ABB RAPID module: Module1_J.mod

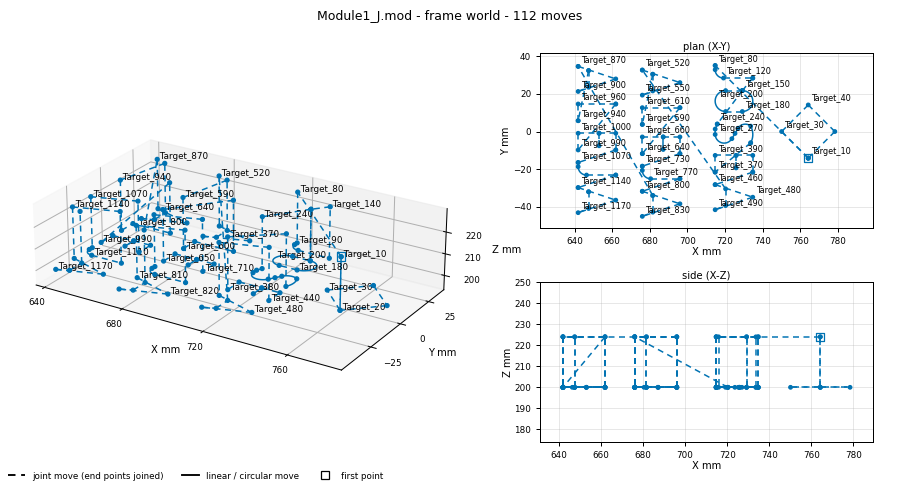
[picture p0: tool path of Module1_J.mod in frame world, 112 of 112 moves have a stored position in this frame; points joined in program order, loops and branches not executed]
MODULE Module1
!Definición de los puntos por donde pasa la trayectoria en forma de robtargets.
!
    CONST robtarget Target_10:=[[149.241,70.858,24],[0.130526196,0,0.991444861,0],[-1,1,-2,0],[9E+09,9E+09,9E+09,9E+09,9E+09,9E+09]];
    CONST robtarget Target_20:=[[149.241,70.858,0],[0.130526196,0,0.991444861,0],[-1,1,-2,0],[9E+09,9E+09,9E+09,9E+09,9E+09,9E+09]];
    CONST robtarget Target_30:=[[135.099,85,0],[0.130526196,0,0.991444861,0],[-1,1,-2,0],[9E+09,9E+09,9E+09,9E+09,9E+09,9E+09]];
    CONST robtarget Target_40:=[[149.241,99.142,0],[0.130526196,0,0.991444861,0],[0,2,-2,0],[9E+09,9E+09,9E+09,9E+09,9E+09,9E+09]];
    CONST robtarget Target_50:=[[163.384,85,0],[0.130526196,0,0.991444861,0],[0,2,-3,0],[9E+09,9E+09,9E+09,9E+09,9E+09,9E+09]];
    CONST robtarget Target_60:=[[149.241,70.858,0],[0.130526196,0,0.991444861,0],[0,2,-3,0],[9E+09,9E+09,9E+09,9E+09,9E+09,9E+09]];
    CONST robtarget Target_70:=[[149.241,70.858,24],[0.130526196,0,0.991444861,0],[-1,1,-2,0],[9E+09,9E+09,9E+09,9E+09,9E+09,9E+09]];
    CONST robtarget Target_80:=[[99.757,120.09,24],[0.130526201,0,0.99144486,-0.000000003],[-1,1,-2,0],[9E+09,9E+09,9E+09,9E+09,9E+09,9E+09]];
    CONST robtarget Target_90:=[[99.757,120.09,0],[0.130526201,0,0.99144486,-0.000000003],[0,2,-3,0],[9E+09,9E+09,9E+09,9E+09,9E+09,9E+09]];
    CONST robtarget Target_100:=[[99.757,117.868,0],[0.130526201,0,0.99144486,-0.000000003],[0,2,-3,0],[9E+09,9E+09,9E+09,9E+09,9E+09,9E+09]];
    CONST robtarget Target_110:=[[101.05812907,114.725008652,0.000349024],[0.130526181,-0.000000019,0.991444863,0.000000016],[0,2,-3,0],[9E+09,9E+09,9E+09,9E+09,9E+09,9E+09]];
    CONST robtarget Target_120:=[[104.201,113.423,0],[0.130526201,0,0.99144486,-0.000000003],[0,2,-3,0],[9E+09,9E+09,9E+09,9E+09,9E+09,9E+09]];
    CONST robtarget Target_130:=[[119.757,113.423,0],[0.130526201,0,0.99144486,-0.000000003],[0,2,-3,0],[9E+09,9E+09,9E+09,9E+09,9E+09,9E+09]];
    CONST robtarget Target_140:=[[119.757,113.423,24],[0.130526201,0,0.99144486,-0.000000003],[0,2,-3,0],[9E+09,9E+09,9E+09,9E+09,9E+09,9E+09]];
    CONST robtarget Target_150:=[[114.201,106.757,24],[0.130526201,0,0.99144486,-0.000000003],[0,2,-3,0],[9E+09,9E+09,9E+09,9E+09,9E+09,9E+09]];
    CONST robtarget Target_160:=[[114.201,106.757,0],[0.130526201,0,0.99144486,-0.000000003],[0,2,-3,0],[9E+09,9E+09,9E+09,9E+09,9E+09,9E+09]];
    CONST robtarget Target_170:=[[119.757,101.201,0],[0.130526201,0,0.99144486,-0.000000003],[0,2,-3,0],[9E+09,9E+09,9E+09,9E+09,9E+09,9E+09]];
    CONST robtarget Target_180:=[[114.201,95.645,0],[0.130526201,0,0.99144486,-0.000000003],[0,2,-3,0],[9E+09,9E+09,9E+09,9E+09,9E+09,9E+09]];
    CONST robtarget Target_190:=[[105.312,95.645,0],[0.130526201,0,0.99144486,-0.000000003],[0,2,-3,0],[9E+09,9E+09,9E+09,9E+09,9E+09,9E+09]];
    CONST robtarget Target_200:=[[99.757,101.201,0],[0.130526201,0,0.99144486,-0.000000003],[0,2,-3,0],[9E+09,9E+09,9E+09,9E+09,9E+09,9E+09]];
    CONST robtarget Target_210:=[[105.312,106.757,0],[0.130526201,0,0.99144486,-0.000000003],[0,2,-3,0],[9E+09,9E+09,9E+09,9E+09,9E+09,9E+09]];
    CONST robtarget Target_220:=[[114.201,106.757,0],[0.130526201,0,0.99144486,-0.000000003],[0,2,-3,0],[9E+09,9E+09,9E+09,9E+09,9E+09,9E+09]];
    CONST robtarget Target_230:=[[114.201,106.757,24],[0.130526201,0,0.99144486,-0.000000003],[0,2,-3,0],[9E+09,9E+09,9E+09,9E+09,9E+09,9E+09]];
    CONST robtarget Target_240:=[[100.868,88.979,24],[0.130526201,0,0.99144486,-0.000000003],[0,2,-3,0],[9E+09,9E+09,9E+09,9E+09,9E+09,9E+09]];
    CONST robtarget Target_250:=[[100.868,88.979,0],[0.130526201,0,0.99144486,-0.000000003],[0,2,-3,0],[9E+09,9E+09,9E+09,9E+09,9E+09,9E+09]];
    CONST robtarget Target_260:=[[99.766,86.31,0],[0.130526201,0,0.99144486,-0.000000003],[0,2,-3,0],[9E+09,9E+09,9E+09,9E+09,9E+09,9E+09]];
    CONST robtarget Target_270:=[[99.757,83.423,0],[0.130526201,0,0.99144486,-0.000000003],[0,2,-3,0],[9E+09,9E+09,9E+09,9E+09,9E+09,9E+09]];
    CONST robtarget Target_280:=[[103.37,78.987,0],[0.130526201,0,0.99144486,-0.000000003],[-1,1,-2,0],[9E+09,9E+09,9E+09,9E+09,9E+09,9E+09]];
    CONST robtarget Target_290:=[[108.646,81.201,0],[0.130526201,0,0.99144486,-0.000000003],[-1,1,-2,0],[9E+09,9E+09,9E+09,9E+09,9E+09,9E+09]];
    CONST robtarget Target_300:=[[110.312,83.979,0],[0.130526201,0,0.99144486,-0.000000003],[-1,1,-2,0],[9E+09,9E+09,9E+09,9E+09,9E+09,9E+09]];
    CONST robtarget Target_310:=[[111.979,86.757,0],[0.130526201,0,0.99144486,-0.000000003],[-1,1,-2,0],[9E+09,9E+09,9E+09,9E+09,9E+09,9E+09]];
    CONST robtarget Target_320:=[[115.054,88.861,0],[0.130526201,0,0.99144486,-0.000000003],[0,2,-3,0],[9E+09,9E+09,9E+09,9E+09,9E+09,9E+09]];
    CONST robtarget Target_340:=[[119.766,83.423,0],[0.130526201,0,0.99144486,-0.000000003],[0,2,-3,0],[9E+09,9E+09,9E+09,9E+09,9E+09,9E+09]];
    CONST robtarget Target_350:=[[118.646,78.979,0],[0.130526201,0,0.99144486,-0.000000003],[-1,1,-2,0],[9E+09,9E+09,9E+09,9E+09,9E+09,9E+09]];
    CONST robtarget Target_360:=[[118.646,78.979,24],[0.130526201,0,0.99144486,-0.000000003],[-1,1,-2,0],[9E+09,9E+09,9E+09,9E+09,9E+09,9E+09]];
    CONST robtarget Target_370:=[[99.757,63.423,24],[0.130526201,0,0.99144486,-0.000000003],[-1,1,-2,0],[9E+09,9E+09,9E+09,9E+09,9E+09,9E+09]];
    CONST robtarget Target_380:=[[99.757,63.423,0],[0.130526201,0,0.99144486,-0.000000003],[-1,1,-2,0],[9E+09,9E+09,9E+09,9E+09,9E+09,9E+09]];
    CONST robtarget Target_390:=[[99.757,72.312,0],[0.130526201,0,0.99144486,-0.000000003],[-1,1,-2,0],[9E+09,9E+09,9E+09,9E+09,9E+09,9E+09]];
    CONST robtarget Target_400:=[[110.868,72.312,0],[0.130526201,0,0.99144486,-0.000000003],[-1,1,-2,0],[9E+09,9E+09,9E+09,9E+09,9E+09,9E+09]];
    CONST robtarget Target_410:=[[110.868,65.645,0],[0.130526201,0,0.99144486,-0.000000003],[-1,1,-2,0],[9E+09,9E+09,9E+09,9E+09,9E+09,9E+09]];
    CONST robtarget Target_420:=[[110.868,72.312,0],[0.130526201,0,0.99144486,-0.000000003],[-1,1,-2,0],[9E+09,9E+09,9E+09,9E+09,9E+09,9E+09]];
    CONST robtarget Target_430:=[[119.757,72.312,0],[0.130526201,0,0.99144486,-0.000000003],[-1,1,-2,0],[9E+09,9E+09,9E+09,9E+09,9E+09,9E+09]];
    CONST robtarget Target_440:=[[119.757,63.423,0],[0.130526201,0,0.99144486,-0.000000003],[-1,1,-2,0],[9E+09,9E+09,9E+09,9E+09,9E+09,9E+09]];
    CONST robtarget Target_450:=[[119.757,63.423,24],[0.130526201,0,0.99144486,-0.000000003],[-1,1,-2,0],[9E+09,9E+09,9E+09,9E+09,9E+09,9E+09]];
    CONST robtarget Target_460:=[[99.757,56.757,24],[0.130526201,0,0.99144486,-0.000000003],[-1,1,-2,0],[9E+09,9E+09,9E+09,9E+09,9E+09,9E+09]];
    CONST robtarget Target_470:=[[99.757,56.757,0],[0.130526201,0,0.99144486,-0.000000003],[-1,1,-2,0],[9E+09,9E+09,9E+09,9E+09,9E+09,9E+09]];
    CONST robtarget Target_480:=[[119.757,50.09,0],[0.130526201,0,0.99144486,-0.000000003],[-1,1,-2,0],[9E+09,9E+09,9E+09,9E+09,9E+09,9E+09]];
    CONST robtarget Target_490:=[[99.757,43.423,0],[0.130526201,0,0.99144486,-0.000000003],[-1,1,-2,0],[9E+09,9E+09,9E+09,9E+09,9E+09,9E+09]];
    CONST robtarget Target_500:=[[105.312,45.645,0],[0.130526201,0,0.99144486,-0.000000003],[-1,1,-2,0],[9E+09,9E+09,9E+09,9E+09,9E+09,9E+09]];
    CONST robtarget Target_510:=[[105.312,54.534,0],[0.130526201,0,0.99144486,-0.000000003],[-1,1,-2,0],[9E+09,9E+09,9E+09,9E+09,9E+09,9E+09]];
    CONST robtarget Target_520:=[[61.026,117.682,24],[0.130526198,0,0.991444861,-0.000000001],[-1,1,-2,0],[9E+09,9E+09,9E+09,9E+09,9E+09,9E+09]];
    CONST robtarget Target_530:=[[61.026,117.682,0],[0.130526198,0,0.991444861,-0.000000001],[0,2,-3,0],[9E+09,9E+09,9E+09,9E+09,9E+09,9E+09]];
    CONST robtarget Target_540:=[[81.026,111.016,0],[0.130526198,0,0.991444861,-0.000000001],[0,2,-3,0],[9E+09,9E+09,9E+09,9E+09,9E+09,9E+09]];
    CONST robtarget Target_550:=[[61.026,104.349,0],[0.130526198,0,0.991444861,-0.000000001],[0,2,-3,0],[9E+09,9E+09,9E+09,9E+09,9E+09,9E+09]];
    CONST robtarget Target_560:=[[66.582,106.571,0],[0.130526198,0,0.991444861,-0.000000001],[0,2,-3,0],[9E+09,9E+09,9E+09,9E+09,9E+09,9E+09]];
    CONST robtarget Target_570:=[[66.582,115.46,0],[0.130526198,0,0.991444861,-0.000000001],[0,2,-3,0],[9E+09,9E+09,9E+09,9E+09,9E+09,9E+09]];
    CONST robtarget Target_580:=[[66.582,115.46,24],[0.130526198,0,0.991444861,-0.000000001],[0,2,-3,0],[9E+09,9E+09,9E+09,9E+09,9E+09,9E+09]];
    CONST robtarget Target_590:=[[61.026,88.794,24],[0.130526198,0,0.991444861,-0.000000001],[0,2,-3,0],[9E+09,9E+09,9E+09,9E+09,9E+09,9E+09]];
    CONST robtarget Target_600:=[[61.026,88.794,0],[0.130526198,0,0.991444861,-0.000000001],[0,2,-3,0],[9E+09,9E+09,9E+09,9E+09,9E+09,9E+09]];
    CONST robtarget Target_610:=[[61.026,97.682,0],[0.130526198,0,0.991444861,-0.000000001],[0,2,-3,0],[9E+09,9E+09,9E+09,9E+09,9E+09,9E+09]];
    CONST robtarget Target_620:=[[81.026,97.682,0],[0.130526198,0,0.991444861,-0.000000001],[0,2,-3,0],[9E+09,9E+09,9E+09,9E+09,9E+09,9E+09]];
    CONST robtarget Target_630:=[[81.026,97.682,24],[0.130526198,0,0.991444861,-0.000000001],[0,2,-3,0],[9E+09,9E+09,9E+09,9E+09,9E+09,9E+09]];
    CONST robtarget Target_640:=[[61.026,73.238,24],[0.130526198,0,0.991444861,-0.000000001],[0,2,-3,0],[9E+09,9E+09,9E+09,9E+09,9E+09,9E+09]];
    CONST robtarget Target_650:=[[61.026,73.238,0],[0.130526198,0,0.991444861,-0.000000001],[-1,1,-2,0],[9E+09,9E+09,9E+09,9E+09,9E+09,9E+09]];
    CONST robtarget Target_660:=[[61.026,82.127,0],[0.130526198,0,0.991444861,-0.000000001],[-1,1,-2,0],[9E+09,9E+09,9E+09,9E+09,9E+09,9E+09]];
    CONST robtarget Target_670:=[[72.137,82.127,0],[0.130526198,0,0.991444861,-0.000000001],[-1,1,-2,0],[9E+09,9E+09,9E+09,9E+09,9E+09,9E+09]];
    CONST robtarget Target_680:=[[72.137,75.46,0],[0.130526198,0,0.991444861,-0.000000001],[-1,1,-2,0],[9E+09,9E+09,9E+09,9E+09,9E+09,9E+09]];
    CONST robtarget Target_690:=[[72.137,82.127,0],[0.130526198,0,0.991444861,-0.000000001],[-1,1,-2,0],[9E+09,9E+09,9E+09,9E+09,9E+09,9E+09]];
    CONST robtarget Target_700:=[[81.026,82.127,0],[0.130526198,0,0.991444861,-0.000000001],[-1,1,-2,0],[9E+09,9E+09,9E+09,9E+09,9E+09,9E+09]];
    CONST robtarget Target_710:=[[81.026,73.238,0],[0.130526198,0,0.991444861,-0.000000001],[-1,1,-2,0],[9E+09,9E+09,9E+09,9E+09,9E+09,9E+09]];
    CONST robtarget Target_720:=[[81.026,73.238,24],[0.130526198,0,0.991444861,-0.000000001],[-1,1,-2,0],[9E+09,9E+09,9E+09,9E+09,9E+09,9E+09]];
    CONST robtarget Target_730:=[[61.026,66.571,24],[0.130526198,0,0.991444861,-0.000000001],[-1,1,-2,0],[9E+09,9E+09,9E+09,9E+09,9E+09,9E+09]];
    CONST robtarget Target_740:=[[61.026,66.571,0],[0.130526198,0,0.991444861,-0.000000001],[-1,1,-2,0],[9E+09,9E+09,9E+09,9E+09,9E+09,9E+09]];
    CONST robtarget Target_750:=[[61.026,64.349,0],[0.130526198,0,0.991444861,-0.000000001],[-1,1,-2,0],[9E+09,9E+09,9E+09,9E+09,9E+09,9E+09]];
    CONST robtarget Target_760:=[[62.328,61.206,0],[0.130526198,0,0.991444861,-0.000000001],[-1,1,-2,0],[9E+09,9E+09,9E+09,9E+09,9E+09,9E+09]];
    CONST robtarget Target_770:=[[65.471,59.905,0],[0.130526198,0,0.991444861,-0.000000001],[-1,1,-2,0],[9E+09,9E+09,9E+09,9E+09,9E+09,9E+09]];
    CONST robtarget Target_780:=[[81.026,59.905,0],[0.130526198,0,0.991444861,-0.000000001],[-1,1,-2,0],[9E+09,9E+09,9E+09,9E+09,9E+09,9E+09]];
    CONST robtarget Target_790:=[[81.026,59.905,24],[0.130526198,0,0.991444861,-0.000000001],[-1,1,-2,0],[9E+09,9E+09,9E+09,9E+09,9E+09,9E+09]];
    CONST robtarget Target_800:=[[61.026,53.238,24],[0.130526198,0,0.991444861,-0.000000001],[-1,1,-2,0],[9E+09,9E+09,9E+09,9E+09,9E+09,9E+09]];
    CONST robtarget Target_810:=[[61.026,53.238,0],[0.130526198,0,0.991444861,-0.000000001],[-1,1,-2,0],[9E+09,9E+09,9E+09,9E+09,9E+09,9E+09]];
    CONST robtarget Target_820:=[[81.026,46.571,0],[0.130526198,0,0.991444861,-0.000000001],[-1,1,-2,0],[9E+09,9E+09,9E+09,9E+09,9E+09,9E+09]];
    CONST robtarget Target_830:=[[61.026,39.905,0],[0.130526198,0,0.991444861,-0.000000001],[-1,1,-2,0],[9E+09,9E+09,9E+09,9E+09,9E+09,9E+09]];
    CONST robtarget Target_840:=[[66.582,42.127,0],[0.130526198,0,0.991444861,-0.000000001],[-1,1,-2,0],[9E+09,9E+09,9E+09,9E+09,9E+09,9E+09]];
    CONST robtarget Target_850:=[[66.582,51.016,0],[0.130526198,0,0.991444861,-0.000000001],[-1,1,-2,0],[9E+09,9E+09,9E+09,9E+09,9E+09,9E+09]];
    CONST robtarget Target_860:=[[66.582,51.016,24],[0.130526198,0,0.991444861,-0.000000001],[-1,1,-2,0],[9E+09,9E+09,9E+09,9E+09,9E+09,9E+09]];
    CONST robtarget Target_870:=[[26.922,119.639,24],[0.130526152,0,0.991444867,0],[-1,1,-2,0],[9E+09,9E+09,9E+09,9E+09,9E+09,9E+09]];
    CONST robtarget Target_880:=[[26.922,119.639,0],[0.130526152,0,0.991444867,0],[0,2,-3,0],[9E+09,9E+09,9E+09,9E+09,9E+09,9E+09]];
    CONST robtarget Target_890:=[[46.922,112.972,0],[0.130526152,0,0.991444867,0],[0,2,-3,0],[9E+09,9E+09,9E+09,9E+09,9E+09,9E+09]];
    CONST robtarget Target_900:=[[26.922,106.305,0],[0.130526152,0,0.991444867,0],[0,2,-3,0],[9E+09,9E+09,9E+09,9E+09,9E+09,9E+09]];
    CONST robtarget Target_910:=[[32.478,108.527,0],[0.130526152,0,0.991444867,0],[0,2,-3,0],[9E+09,9E+09,9E+09,9E+09,9E+09,9E+09]];
    CONST robtarget Target_920:=[[32.478,117.416,0],[0.130526152,0,0.991444867,0],[0,2,-3,0],[9E+09,9E+09,9E+09,9E+09,9E+09,9E+09]];
    CONST robtarget Target_930:=[[32.478,117.416,24],[0.130526152,0,0.991444867,0],[0,2,-3,0],[9E+09,9E+09,9E+09,9E+09,9E+09,9E+09]];
    CONST robtarget Target_940:=[[26.922,90.75,24],[0.130526152,0,0.991444867,0],[0,2,-3,0],[9E+09,9E+09,9E+09,9E+09,9E+09,9E+09]];
    CONST robtarget Target_950:=[[26.922,90.75,0],[0.130526152,0,0.991444867,0],[0,2,-3,0],[9E+09,9E+09,9E+09,9E+09,9E+09,9E+09]];
    CONST robtarget Target_960:=[[26.922,99.639,0],[0.130526152,0,0.991444867,0],[0,2,-3,0],[9E+09,9E+09,9E+09,9E+09,9E+09,9E+09]];
    CONST robtarget Target_970:=[[46.922,99.639,0],[0.130526152,0,0.991444867,0],[0,2,-3,0],[9E+09,9E+09,9E+09,9E+09,9E+09,9E+09]];
    CONST robtarget Target_980:=[[46.922,99.639,24],[0.130526152,0,0.991444867,0],[0,2,-3,0],[9E+09,9E+09,9E+09,9E+09,9E+09,9E+09]];
    CONST robtarget Target_990:=[[26.922,75.194,0],[0.130526152,0,0.991444867,0],[0,2,-3,0],[9E+09,9E+09,9E+09,9E+09,9E+09,9E+09]];
    CONST robtarget Target_1000:=[[26.922,84.083,0],[0.130526152,0,0.991444867,0],[-1,1,-2,0],[9E+09,9E+09,9E+09,9E+09,9E+09,9E+09]];
    CONST robtarget Target_1010:=[[38.033,84.083,0],[0.130526152,0,0.991444867,0],[-1,1,-2,0],[9E+09,9E+09,9E+09,9E+09,9E+09,9E+09]];
    CONST robtarget Target_1020:=[[38.033,77.416,0],[0.130526152,0,0.991444867,0],[-1,1,-2,0],[9E+09,9E+09,9E+09,9E+09,9E+09,9E+09]];
    CONST robtarget Target_1030:=[[38.033,84.083,0],[0.130526152,0,0.991444867,0],[-1,1,-2,0],[9E+09,9E+09,9E+09,9E+09,9E+09,9E+09]];
    CONST robtarget Target_1040:=[[46.922,84.083,0],[0.130526152,0,0.991444867,0],[-1,1,-2,0],[9E+09,9E+09,9E+09,9E+09,9E+09,9E+09]];
    CONST robtarget Target_1050:=[[46.922,75.194,0],[0.130526152,0,0.991444867,0],[-1,1,-2,0],[9E+09,9E+09,9E+09,9E+09,9E+09,9E+09]];
    CONST robtarget Target_1060:=[[46.922,75.194,24],[0.130526152,0,0.991444867,0],[-1,1,-2,0],[9E+09,9E+09,9E+09,9E+09,9E+09,9E+09]];
    CONST robtarget Target_1070:=[[26.922,68.527,24],[0.130526152,0,0.991444867,0],[-1,1,-2,0],[9E+09,9E+09,9E+09,9E+09,9E+09,9E+09]];
    CONST robtarget Target_1080:=[[26.922,68.527,0],[0.130526152,0,0.991444867,0],[-1,1,-2,0],[9E+09,9E+09,9E+09,9E+09,9E+09,9E+09]];
    CONST robtarget Target_1090:=[[26.922,66.305,0],[0.130526152,0,0.991444867,0],[-1,1,-2,0],[9E+09,9E+09,9E+09,9E+09,9E+09,9E+09]];
    CONST robtarget Target_1100:=[[28.224,63.163,0],[0.130526152,0,0.991444867,0],[-1,1,-2,0],[9E+09,9E+09,9E+09,9E+09,9E+09,9E+09]];
    CONST robtarget Target_1110:=[[31.367,61.861,0],[0.130526152,0,0.991444867,0],[-1,1,-2,0],[9E+09,9E+09,9E+09,9E+09,9E+09,9E+09]];
    CONST robtarget Target_1120:=[[46.922,61.861,0],[0.130526152,0,0.991444867,0],[-1,1,-2,0],[9E+09,9E+09,9E+09,9E+09,9E+09,9E+09]];
    CONST robtarget Target_1130:=[[46.922,61.861,24],[0.130526152,0,0.991444867,0],[-1,1,-2,0],[9E+09,9E+09,9E+09,9E+09,9E+09,9E+09]];
    CONST robtarget Target_1140:=[[26.922,55.194,24],[0.130526152,0,0.991444867,0],[-1,1,-2,0],[9E+09,9E+09,9E+09,9E+09,9E+09,9E+09]];
    CONST robtarget Target_1150:=[[26.922,55.194,0],[0.130526152,0,0.991444867,0],[-1,1,-2,0],[9E+09,9E+09,9E+09,9E+09,9E+09,9E+09]];
    CONST robtarget Target_1160:=[[46.922,48.527,0],[0.130526152,0,0.991444867,0],[-1,1,-2,0],[9E+09,9E+09,9E+09,9E+09,9E+09,9E+09]];
    CONST robtarget Target_1170:=[[26.922,41.861,0],[0.130526152,0,0.991444867,0],[-1,1,-2,0],[9E+09,9E+09,9E+09,9E+09,9E+09,9E+09]];
    CONST robtarget Target_1180:=[[32.478,44.083,0],[0.130526152,0,0.991444867,0],[-1,1,-2,0],[9E+09,9E+09,9E+09,9E+09,9E+09,9E+09]];
    CONST robtarget Target_1190:=[[32.478,52.972,0],[0.130526152,0,0.991444867,0],[-1,1,-2,0],[9E+09,9E+09,9E+09,9E+09,9E+09,9E+09]];
    CONST robtarget Target_1200:=[[32.478,52.972,24],[0.130526152,0,0.991444867,0],[-1,1,-2,0],[9E+09,9E+09,9E+09,9E+09,9E+09,9E+09]];
    CONST robtarget Target_330:=[[118.646,87.868,0],[0.130526201,0,0.99144486,-0.000000003],[0,2,-3,0],[9E+09,9E+09,9E+09,9E+09,9E+09,9E+09]];
!Definición del objeto tooldata con los dato de la herramienta a usar en el efector final del robot.
!
    PERS tooldata MyNewTool:=[TRUE,[[25.289,0,191.739],[0.923879533,0,0.382683432,0]],[0.5,[-37.543,-11.677,118.601],[1,0,0,0],0,0,0]];
!Definición del objeto wobjdata con los datos del WorkObject donde el robot va a trazar la trayectoria.
!Entonces si se necesita girar o modificar la trayectoria simplemente se modifica los datos del workobject.
!
    TASK PERS wobjdata Workobject_1:=[FALSE,TRUE,"",[[615,-85,200],[1,0,0,0]],[[0,0,0],[1,0,0,0]]];
!Proceso que contiene las instrucciones de movimiento del robot
!
    PROC Path_10()
!La instrucción MoveJ se utiliza ya que esto permite al robot trabajar en el espacio articular.
!Esto permite que incluso si la trayectoria se rota, el robot so sufrirá de errores de singularidad a causa de gimbal locking.
!
!Se utiliza la Instrucción MoveC para definir las trayectorias curvas de algunas de las letras del logo.
!Se tuvo mucho cuidado de evitar las curvas que generasen errores como círculo indefinidos o puntos inalcanzables.
!
        MoveJ Target_10,v100,fine,MyNewTool\WObj:=Workobject_1;
        MoveJ Target_20,v100,z10,MyNewTool\WObj:=Workobject_1;
        MoveJ Target_30,v100,z10,MyNewTool\WObj:=Workobject_1;
        MoveJ Target_40,v100,z10,MyNewTool\WObj:=Workobject_1;
        MoveJ Target_50,v100,z10,MyNewTool\WObj:=Workobject_1;
        MoveJ Target_60,v100,z10,MyNewTool\WObj:=Workobject_1;
        MoveJ Target_70,v100,z10,MyNewTool\WObj:=Workobject_1;
        MoveJ Target_80,v100,fine,MyNewTool\WObj:=Workobject_1;
        MoveJ Target_90,v100,z10,MyNewTool\WObj:=Workobject_1;
        MoveJ Target_100,v100,z10,MyNewTool\WObj:=Workobject_1;
        MoveC Target_110,Target_120,v100,z10,MyNewTool\WObj:=Workobject_1;
        MoveJ Target_130,v100,z10,MyNewTool\WObj:=Workobject_1;
        MoveJ Target_140,v100,z10,MyNewTool\WObj:=Workobject_1;
        MoveJ Target_150,v100,z10,MyNewTool\WObj:=Workobject_1;
        MoveJ Target_160,v100,z10,MyNewTool\WObj:=Workobject_1;
        MoveC Target_170,Target_180,v100,z10,MyNewTool\WObj:=Workobject_1;
        MoveJ Target_190,v100,z10,MyNewTool\WObj:=Workobject_1;
        MoveC Target_200,Target_210,v100,z10,MyNewTool\WObj:=Workobject_1;
        MoveJ Target_220,v100,z10,MyNewTool\WObj:=Workobject_1;
        MoveJ Target_230,v100,z10,MyNewTool\WObj:=Workobject_1;
        MoveJ Target_240,v100,z10,MyNewTool\WObj:=Workobject_1;
        MoveJ Target_250,v100,z10,MyNewTool\WObj:=Workobject_1;
        MoveJ Target_260,v100,z10,MyNewTool\WObj:=Workobject_1;
        MoveJ Target_270,v100,z10,MyNewTool\WObj:=Workobject_1;
        MoveC Target_280,Target_290,v100,z10,MyNewTool\WObj:=Workobject_1;
        MoveJ Target_300,v100,z10,MyNewTool\WObj:=Workobject_1;
        MoveJ Target_310,v100,z10,MyNewTool\WObj:=Workobject_1;
        MoveC Target_320,Target_330,v100,z10,MyNewTool\WObj:=Workobject_1;
        MoveC Target_340,Target_350,v100,z10,MyNewTool\WObj:=Workobject_1;
        MoveJ Target_360,v100,z10,MyNewTool\WObj:=Workobject_1;
        MoveJ Target_370,v100,z10,MyNewTool\WObj:=Workobject_1;
        MoveJ Target_380,v100,z10,MyNewTool\WObj:=Workobject_1;
        MoveJ Target_390,v100,z10,MyNewTool\WObj:=Workobject_1;
        MoveJ Target_400,v100,z10,MyNewTool\WObj:=Workobject_1;
        MoveJ Target_410,v100,z10,MyNewTool\WObj:=Workobject_1;
        MoveJ Target_420,v100,z10,MyNewTool\WObj:=Workobject_1;
        MoveJ Target_430,v100,z10,MyNewTool\WObj:=Workobject_1;
        MoveJ Target_440,v100,z10,MyNewTool\WObj:=Workobject_1;
        MoveJ Target_450,v100,z10,MyNewTool\WObj:=Workobject_1;
        MoveJ Target_460,v100,z10,MyNewTool\WObj:=Workobject_1;
        MoveJ Target_470,v100,z10,MyNewTool\WObj:=Workobject_1;
        MoveJ Target_480,v100,z10,MyNewTool\WObj:=Workobject_1;
        MoveJ Target_490,v100,z10,MyNewTool\WObj:=Workobject_1;
        MoveJ Target_500,v100,z10,MyNewTool\WObj:=Workobject_1;
        MoveJ Target_510,v100,z10,MyNewTool\WObj:=Workobject_1;
        MoveJ Target_520,v100,fine,MyNewTool\WObj:=Workobject_1;
        MoveJ Target_530,v100,z10,MyNewTool\WObj:=Workobject_1;
        MoveJ Target_540,v100,z10,MyNewTool\WObj:=Workobject_1;
        MoveJ Target_550,v100,z10,MyNewTool\WObj:=Workobject_1;
        MoveJ Target_560,v100,z10,MyNewTool\WObj:=Workobject_1;
        MoveJ Target_570,v100,z10,MyNewTool\WObj:=Workobject_1;
        MoveJ Target_580,v100,z10,MyNewTool\WObj:=Workobject_1;
        MoveJ Target_590,v100,z10,MyNewTool\WObj:=Workobject_1;
        MoveJ Target_600,v100,z10,MyNewTool\WObj:=Workobject_1;
        MoveJ Target_610,v100,z10,MyNewTool\WObj:=Workobject_1;
        MoveJ Target_620,v100,z10,MyNewTool\WObj:=Workobject_1;
        MoveJ Target_630,v100,z10,MyNewTool\WObj:=Workobject_1;
        MoveJ Target_640,v100,z10,MyNewTool\WObj:=Workobject_1;
        MoveJ Target_650,v100,z10,MyNewTool\WObj:=Workobject_1;
        MoveJ Target_660,v100,z10,MyNewTool\WObj:=Workobject_1;
        MoveJ Target_670,v100,z10,MyNewTool\WObj:=Workobject_1;
        MoveJ Target_680,v100,z10,MyNewTool\WObj:=Workobject_1;
        MoveJ Target_690,v100,z10,MyNewTool\WObj:=Workobject_1;
        MoveJ Target_700,v100,z10,MyNewTool\WObj:=Workobject_1;
        MoveJ Target_710,v100,z10,MyNewTool\WObj:=Workobject_1;
        MoveJ Target_720,v100,z10,MyNewTool\WObj:=Workobject_1;
        MoveJ Target_730,v100,z10,MyNewTool\WObj:=Workobject_1;
        MoveJ Target_740,v100,z10,MyNewTool\WObj:=Workobject_1;
        MoveJ Target_750,v100,z10,MyNewTool\WObj:=Workobject_1;
        MoveC Target_760,Target_770,v100,z10,MyNewTool\WObj:=Workobject_1;
        MoveJ Target_780,v100,z10,MyNewTool\WObj:=Workobject_1;
        MoveJ Target_790,v100,z10,MyNewTool\WObj:=Workobject_1;
        MoveJ Target_800,v100,z10,MyNewTool\WObj:=Workobject_1;
        MoveJ Target_810,v100,z10,MyNewTool\WObj:=Workobject_1;
        MoveJ Target_820,v100,z10,MyNewTool\WObj:=Workobject_1;
        MoveJ Target_830,v100,z10,MyNewTool\WObj:=Workobject_1;
        MoveJ Target_840,v100,z10,MyNewTool\WObj:=Workobject_1;
        MoveJ Target_850,v100,z10,MyNewTool\WObj:=Workobject_1;
        MoveJ Target_860,v100,z10,MyNewTool\WObj:=Workobject_1;
        MoveJ Target_870,v100,fine,MyNewTool\WObj:=Workobject_1;
        MoveJ Target_880,v100,z10,MyNewTool\WObj:=Workobject_1;
        MoveJ Target_890,v100,z10,MyNewTool\WObj:=Workobject_1;
        MoveJ Target_900,v100,z10,MyNewTool\WObj:=Workobject_1;
        MoveJ Target_910,v100,z10,MyNewTool\WObj:=Workobject_1;
        MoveJ Target_920,v100,z10,MyNewTool\WObj:=Workobject_1;
        MoveJ Target_930,v100,z10,MyNewTool\WObj:=Workobject_1;
        MoveJ Target_940,v100,z10,MyNewTool\WObj:=Workobject_1;
        MoveJ Target_950,v100,z10,MyNewTool\WObj:=Workobject_1;
        MoveJ Target_960,v100,z10,MyNewTool\WObj:=Workobject_1;
        MoveJ Target_970,v100,z10,MyNewTool\WObj:=Workobject_1;
        MoveJ Target_980,v100,z10,MyNewTool\WObj:=Workobject_1;
        MoveJ Target_990,v100,z10,MyNewTool\WObj:=Workobject_1;
        MoveJ Target_1000,v100,z10,MyNewTool\WObj:=Workobject_1;
        MoveJ Target_1010,v100,z10,MyNewTool\WObj:=Workobject_1;
        MoveJ Target_1020,v100,z10,MyNewTool\WObj:=Workobject_1;
        MoveJ Target_1030,v100,z10,MyNewTool\WObj:=Workobject_1;
        MoveJ Target_1040,v100,z10,MyNewTool\WObj:=Workobject_1;
        MoveJ Target_1050,v100,z10,MyNewTool\WObj:=Workobject_1;
        MoveJ Target_1060,v100,z10,MyNewTool\WObj:=Workobject_1;
        MoveJ Target_1070,v100,z10,MyNewTool\WObj:=Workobject_1;
        MoveJ Target_1080,v100,z10,MyNewTool\WObj:=Workobject_1;
        MoveJ Target_1090,v100,z10,MyNewTool\WObj:=Workobject_1;
        MoveC Target_1100,Target_1110,v100,z10,MyNewTool\WObj:=Workobject_1;
        MoveJ Target_1120,v100,z10,MyNewTool\WObj:=Workobject_1;
        MoveJ Target_1130,v100,z10,MyNewTool\WObj:=Workobject_1;
        MoveJ Target_1140,v100,z10,MyNewTool\WObj:=Workobject_1;
        MoveJ Target_1150,v100,z10,MyNewTool\WObj:=Workobject_1;
        MoveJ Target_1160,v100,z10,MyNewTool\WObj:=Workobject_1;
        MoveJ Target_1170,v100,z10,MyNewTool\WObj:=Workobject_1;
        MoveJ Target_1180,v100,z10,MyNewTool\WObj:=Workobject_1;
        MoveJ Target_1190,v100,z10,MyNewTool\WObj:=Workobject_1;
        MoveJ Target_1200,v100,z10,MyNewTool\WObj:=Workobject_1;
    ENDPROC
ENDMODULE
